// TIA Portal V18 export
// export: Created 2025-12-01T12:37:58.069048Z, ExportSetting None, DisplayName Totally Integrated Automation Portal, DisplayVersion V18 Update 5, DisplayName TIA Portal Openness, DisplayVersion V18 Update 5, DisplayName TIA Portal Teamcenter Gateway, DisplayVersion V18, DisplayName TIA Portal Version Control Interface, DisplayVersion V18, DisplayName STEP 7 Professional, DisplayVersion V18 Update 5, DisplayName STEP 7 Safety, DisplayVersion V18, DisplayName WinCC Professional, DisplayVersion V18 Update 5
ORGANIZATION_BLOCK "02_Warm Restart"   // OB100, LAD, Startup
TITLE = "Complete Restart"
{ S7_Optimized_Access := 'FALSE' }
AUTHOR : RCS
// 1.该部分用户可以根据系统的需要将CPU第一次扫描需要执行的逻辑写在此处
// stored: AutoNumber false, SetENOAutomatically false
   VAR_TEMP
      OB100_EV_CLASS : Byte;   // 16#13, Event class 1, Entering event state, Event logged in diagnostic buffer
      OB100_STRTUP : Byte;   // 16#81/82/83/84 Method of startup
      OB100_PRIORITY : Byte;   // Priority of OB Execution
      OB100_OB_NUMBR : Byte;   // 100 (Organization block 100, OB100)
      OB100_RESERVED_1 : Byte;   // Reserved for system
      OB100_RESERVED_2 : Byte;   // Reserved for system
      OB100_STOP : Word;   // Event that caused CPU to stop (16#4xxx)
      OB100_STRT_INFO : DWord;   // Information on how system started
      OB100_DATE_TIME : Date_And_Time;   // Date and time OB100 started
   END_VAR
BEGIN

REGION Network 1
   // 系统程序段无需改动
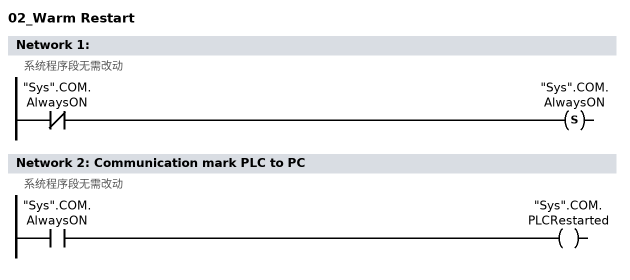
   RUNG wire#powerrail
      I_Contact( "Sys".COM.AlwaysON )
      S_Coil( "Sys".COM.AlwaysON )
   END_RUNG
   // the same network as SCL:
   IF NOT "Sys".COM.AlwaysON THEN "Sys".COM.AlwaysON := TRUE; END_IF;
END_REGION

REGION Network 2: Communication mark PLC to PC
   // 系统程序段无需改动
   RUNG wire#powerrail
      Contact( "Sys".COM.AlwaysON )
      Coil( "Sys".COM.PLCRestarted )
   END_RUNG
   // the same network as SCL:
   "Sys".COM.PLCRestarted := "Sys".COM.AlwaysON;
END_REGION

NETWORK
TITLE = 

      L     1;
      T     "Station_Sys".Status.ModeSV;

END_ORGANIZATION_BLOCK
